// Mitsubishi GX Works2 project: 0723_2번정지추가완료   PLC: Q02/Q02H

PROGRAM MAIN
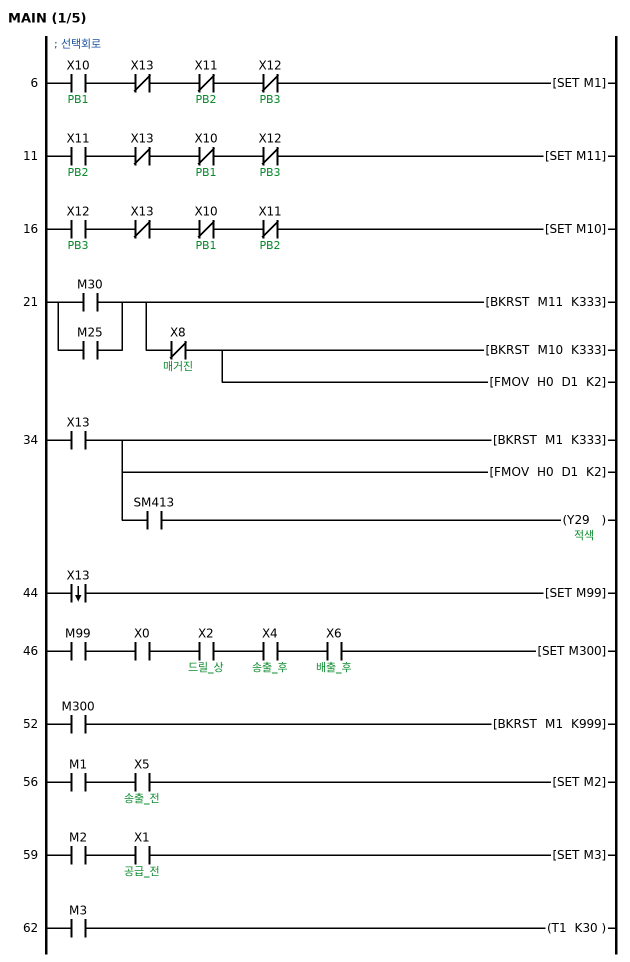
; 선택회로
6     LD      X10  ; PB1
      ANI     X13
      ANI     X11  ; PB2
      ANI     X12  ; PB3
      SET     M1
11    LD      X11  ; PB2
      ANI     X13
      ANI     X10  ; PB1
      ANI     X12  ; PB3
      SET     M11
16    LD      X12  ; PB3
      ANI     X13
      ANI     X10  ; PB1
      ANI     X11  ; PB2
      SET     M10
21    LD      M30
      OR      M25
      BKRST   M11 K333
      ANI     X8  ; 매거진
      BKRST   M10 K333
      FMOV    H0 D1 K2
34    LD      X13
      BKRST   M1 K333
      FMOV    H0 D1 K2
      AND     SM413
      OUT     Y29  ; 적색
44    LDF     X13
      SET     M99
46    LD      M99
      AND     X0
      AND     X2  ; 드릴_상
      AND     X4  ; 송출_후
      AND     X6  ; 배출_후
      SET     M300
52    LD      M300
      BKRST   M1 K999
56    LD      M1
      AND     X5  ; 송출_전
      SET     M2
59    LD      M2
      AND     X1  ; 공급_전
      SET     M3
62    LD      M3
      OUT     T1 K30
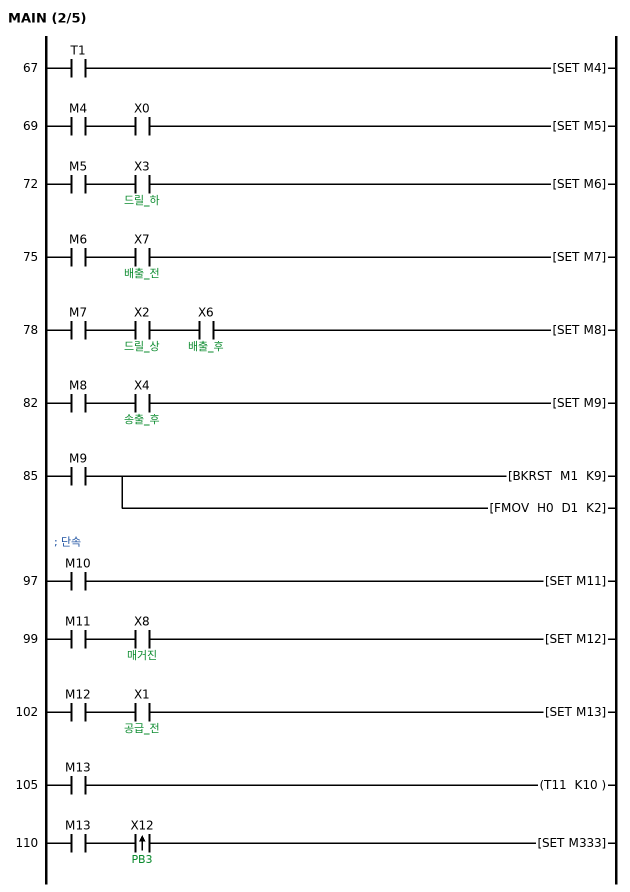
67    LD      T1
      SET     M4
69    LD      M4
      AND     X0
      SET     M5
72    LD      M5
      AND     X3  ; 드릴_하
      SET     M6
75    LD      M6
      AND     X7  ; 배출_전
      SET     M7
78    LD      M7
      AND     X2  ; 드릴_상
      AND     X6  ; 배출_후
      SET     M8
82    LD      M8
      AND     X4  ; 송출_후
      SET     M9
85    LD      M9
      BKRST   M1 K9
      FMOV    H0 D1 K2
; 단속
97    LD      M10
      SET     M11
99    LD      M11
      AND     X8  ; 매거진
      SET     M12
102   LD      M12
      AND     X1  ; 공급_전
      SET     M13
105   LD      M13
      OUT     T11 K10
110   LD      M13
      ANDP    X12  ; PB3
      SET     M333
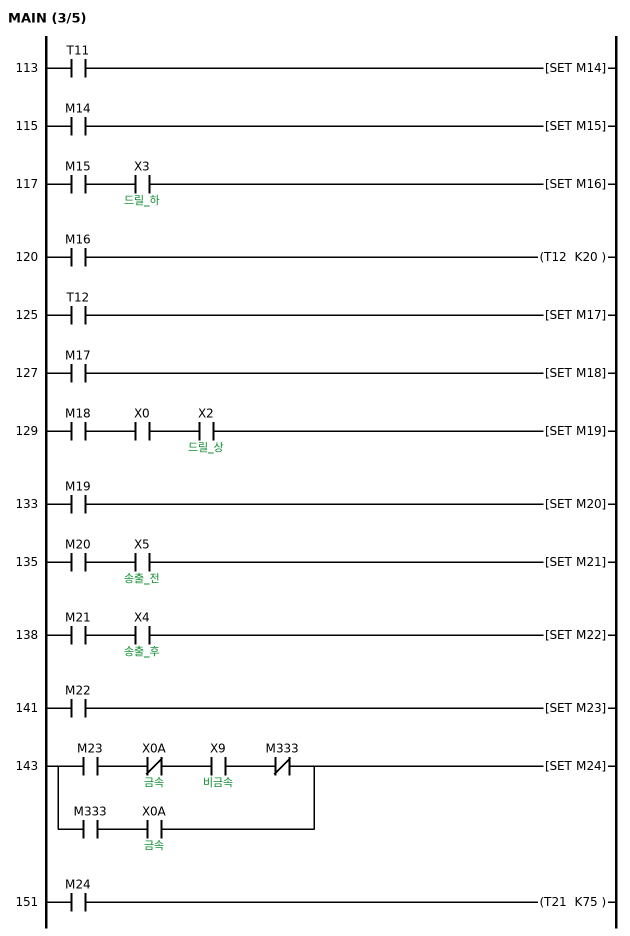
113   LD      T11
      SET     M14
115   LD      M14
      SET     M15
117   LD      M15
      AND     X3  ; 드릴_하
      SET     M16
120   LD      M16
      OUT     T12 K20
125   LD      T12
      SET     M17
127   LD      M17
      SET     M18
129   LD      M18
      AND     X0
      AND     X2  ; 드릴_상
      SET     M19
133   LD      M19
      SET     M20
135   LD      M20
      AND     X5  ; 송출_전
      SET     M21
138   LD      M21
      AND     X4  ; 송출_후
      SET     M22
141   LD      M22
      SET     M23
143   LD      M23
      ANI     X0A  ; 금속
      AND     X9  ; 비금속
      ANI     M333
      LD      M333
      AND     X0A  ; 금속
      ORB
      SET     M24
151   LD      M24
      OUT     T21 K75
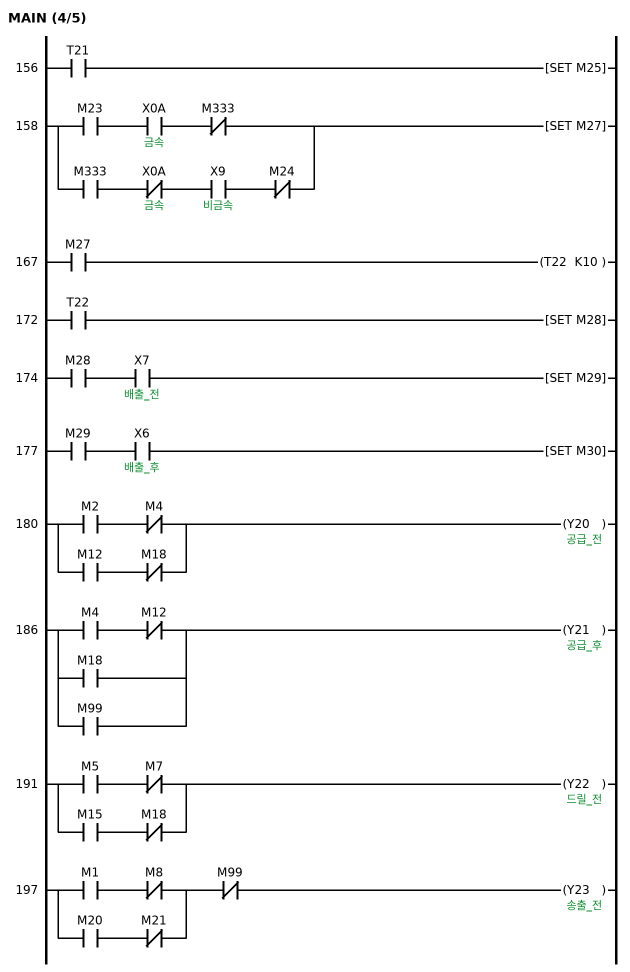
156   LD      T21
      SET     M25
158   LD      M23
      AND     X0A  ; 금속
      ANI     M333
      LD      M333
      ANI     X0A  ; 금속
      AND     X9  ; 비금속
      ANI     M24
      ORB
      SET     M27
167   LD      M27
      OUT     T22 K10
172   LD      T22
      SET     M28
174   LD      M28
      AND     X7  ; 배출_전
      SET     M29
177   LD      M29
      AND     X6  ; 배출_후
      SET     M30
180   LD      M2
      ANI     M4
      LD      M12
      ANI     M18
      ORB
      OUT     Y20  ; 공급_전
186   LD      M4
      ANI     M12
      OR      M18
      OR      M99
      OUT     Y21  ; 공급_후
191   LD      M5
      ANI     M7
      LD      M15
      ANI     M18
      ORB
      OUT     Y22  ; 드릴_전
197   LD      M1
      ANI     M8
      LD      M20
      ANI     M21
      ORB
      ANI     M99
      OUT     Y23  ; 송출_전
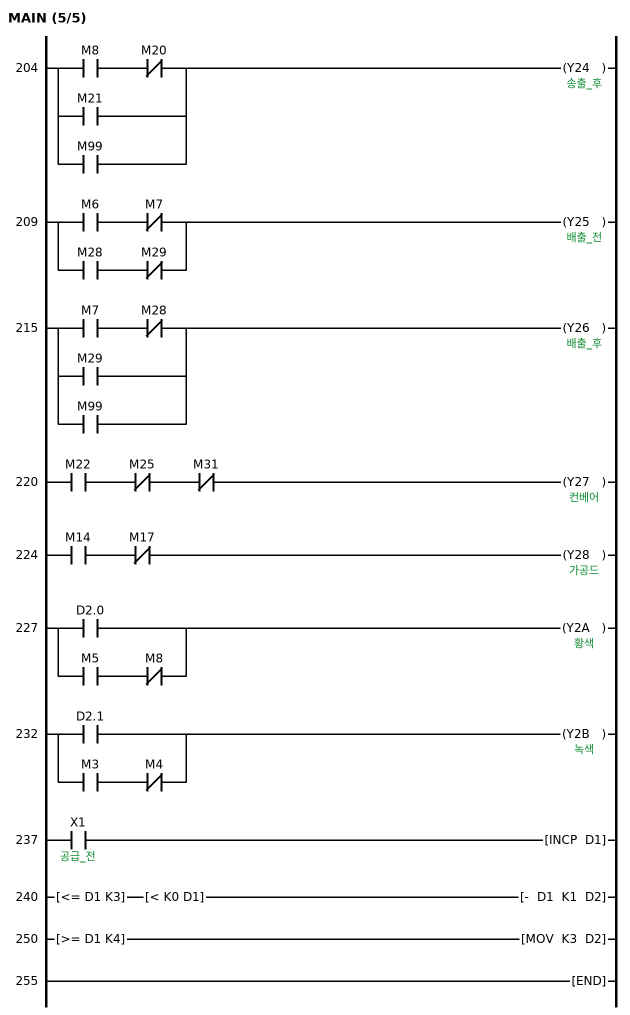
204   LD      M8
      ANI     M20
      OR      M21
      OR      M99
      OUT     Y24  ; 송출_후
209   LD      M6
      ANI     M7
      LD      M28
      ANI     M29
      ORB
      OUT     Y25  ; 배출_전
215   LD      M7
      ANI     M28
      OR      M29
      OR      M99
      OUT     Y26  ; 배출_후
220   LD      M22
      ANI     M25
      ANI     M31
      OUT     Y27  ; 컨베어
224   LD      M14
      ANI     M17
      OUT     Y28  ; 가공드
227   LD      D2.0
      LD      M5
      ANI     M8
      ORB
      OUT     Y2A  ; 황색
232   LD      D2.1
      LD      M3
      ANI     M4
      ORB
      OUT     Y2B  ; 녹색
237   LD      X1  ; 공급_전
      INCP    D1
240   LD<=    D1 K3
      AND<    K0 D1
      -       D1 K1 D2
250   LD>=    D1 K4
      MOV     K3 D2
255   END
END_PROGRAM
